FUNCTION_BLOCK POU_TestGit1
VAR_INPUT
END_VAR
VAR_OUTPUT
END_VAR
VAR
END_VAR

END_FUNCTION_BLOCK

(* stored: Version 1.1.0.1, ProductVersion 3.1.4024.11
   POU POU_TestGit1: Id {828f58be-d085-42d5-9082-bf4494704488}, SpecialFunc None *)
